// TIA Portal V19 export
TYPE "Motor2Ctrl"
// stored: Access Published
   STRUCT
      SafeStop : Bool;
      Rst : Bool;   // Reset alarms command
      RunBkw : Bool;   // Command:
      RunFwd : Bool;   // Command:
   END_STRUCT;
END_TYPE
